FUNCTION_BLOCK FB_FIFO
VAR_INPUT
END_VAR
VAR_OUTPUT
END_VAR
VAR
	fbfifo : FB_FIFO_OOP;
END_VAR

//FB_Init is always available implicitly and it is used primarily for initialization.
//The return value is not evaluated. For a specific influence, you can also declare the
//methods explicitly and provide additional code there with the standard initialization
//code. You can evaluate the return value.
METHOD FB_Init: BOOL
VAR_INPUT
    bInitRetains: BOOL; // TRUE: the retain variables are initialized (reset warm / reset cold)
    bInCopyCode: BOOL;  // TRUE: the instance will be copied to the copy code afterward (online change)   
END_VAR
THIS^.fbfifo.Init(-3);
END_METHOD

PROPERTY ifEmptyRegister : IF_EmptyRegister
GET
ifEmptyRegister :=THIS^.fbfifo;
END_GET
END_PROPERTY

PROPERTY ifFillRegister : IF_FillRegister
GET
ifEmptyRegister := THIS^.ifFillRegister;
END_GET
END_PROPERTY

PROPERTY ifRegister : IF_Register
GET
ifRegister:=THIS^.fbfifo;
END_GET
END_PROPERTY

END_FUNCTION_BLOCK

(* stored: Version 1.1.0.1
   POU FB_FIFO: Id {1c6a94ff-259f-4eba-af26-5235703782a8}, SpecialFunc None
   Method FB_Init: Id {8db51797-4263-4cbb-a612-38cb41f7acf8}
   Property ifEmptyRegister: Id {acf42f43-b488-4f05-8ff7-200670a88927}
   Get Get: Id {e6828dd7-f8e1-4f19-a6e0-9c09bc5b44ce}
   Property ifFillRegister: Id {2f354821-bac2-460a-af1f-f7254a3ff9df}
   Get Get: Id {a1caffc7-1ba1-4d71-b9a3-37cf9dd05a8f}
   Property ifRegister: Id {fef76588-1cba-4a4c-88e2-1c58ff997c82}
   Get Get: Id {b8e41cd3-0b67-4f74-8bbf-1b111e54c3ee} *)
